(* PLC project VisuTest.project, CODESYS CODESYS V3.5 SP17 Patch 2 *)
(* stored: creationDateTime 2022-02-17T09:26:16.669529, modificationDateTime 2022-02-16T16:05:59.7420926 *)

TYPE DUT : STRUCT

END_STRUCT;
END_TYPE

PROGRAM PLC_PRG

END_PROGRAM

FUNCTION_BLOCK POU

END_FUNCTION_BLOCK

CONFIGURATION Device
  RESOURCE Application ON PLC
    TASK MainTask(INTERVAL := T#20ms, PRIORITY := 1);
    TASK VISU_TASK(INTERVAL := T#100ms, PRIORITY := 31);
    TASK Task(INTERVAL := T#20ms, PRIORITY := 1);
    PROGRAM PLC_PRG WITH MainTask : PLC_PRG;
    PROGRAM VisuElems.Visu_Prg WITH VISU_TASK : VisuElems.Visu_Prg;
  END_RESOURCE
END_CONFIGURATION
